(* Logix 5000 project; controller CLASE_1 Emulate 5570 rev 28.11; software revision 28.02; part 7 of 15 *)
(* tags used below, declared in another part *)
   Inp_OvrdCmd : DINT;   // Override Mode Command: 0=None, 1=Stop, 2=Start
   PCmd_Start : BOOL;   // Program Command to Start Motor
   PCmd_Stop : BOOL;   // Program Command to Stop Motor
   OCmd_Start : BOOL;   // Operator Command to Start Motor
   OCmd_Stop : BOOL;   // Operator Command to Stop Motor
   Out_Run : BOOL;   // 1=Run Motor, 0=Stop Motor
   Out_Start : BOOL;   // 1=Start Motor, 0=Motor left in current state
   Out_Stop : BOOL;   // 1=Stop Motor, 0=Motor left in current state
   Val_Cmd : SINT;   // Device Command 0=None, 1=Stop, 2=Start
   Nrdy_OperPrio : BOOL;   // 1=Device Not Ready: Operator State 0 Priority Command Requires Reset
   Nrdy_Fail : BOOL;   // 1=Device Not Ready: Device Failure (Shed Requires Reset)
   P_Motor : BOOL;   // Unique Parameter Name for auto - discovery
   Wrk_Run : BOOL;   // 1=Motor should be "running", 0=should be "stopped"
   Wrk_RunFdbk : BOOL;   // Run Feedback based on mode, simulation, etc. 1=running
(* P_Motor, continued *)

ROUTINE Prescan   (* ladder *)
// Clear Ownership, clear "lurking" Commands
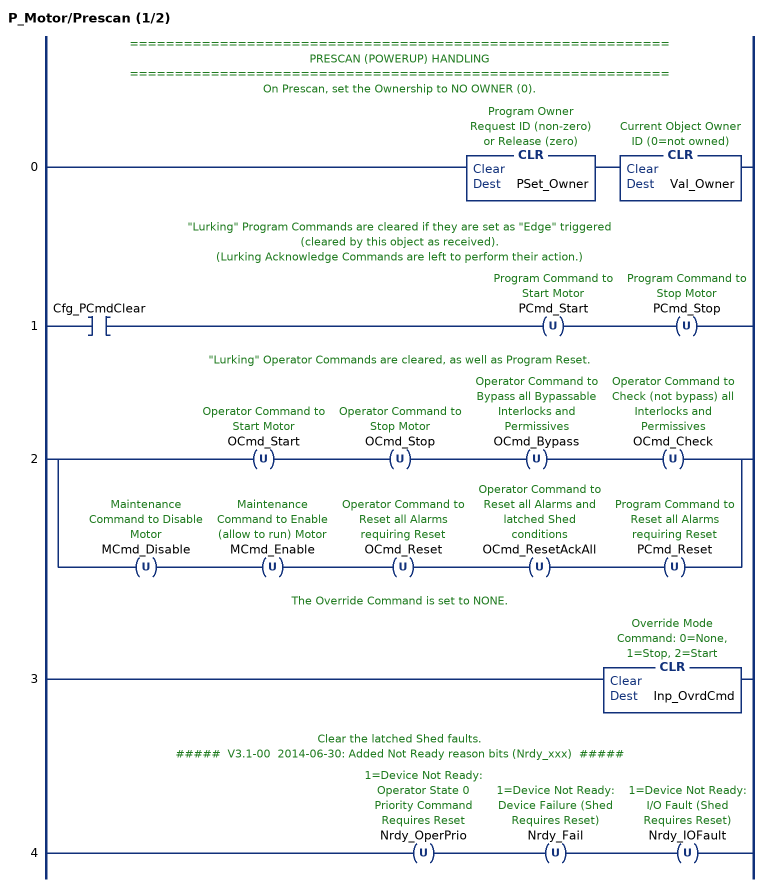
   // ============================================================
   // PRESCAN (POWERUP) HANDLING
   // ============================================================
   // On Prescan, set the Ownership to NO OWNER (0).
   0: CLR(PSet_Owner)CLR(Val_Owner);
   // "Lurking" Program Commands are cleared if they are set as "Edge" triggered
   // (cleared by this object as received).
   // (Lurking Acknowledge Commands are left to perform their action.)
   1: XIC(Cfg_PCmdClear)OTU(PCmd_Start)OTU(PCmd_Stop);
   // "Lurking" Operator Commands are cleared, as well as Program Reset.
   2: [OTU(OCmd_Start) OTU(OCmd_Stop) OTU(OCmd_Bypass) OTU(OCmd_Check) ,OTU(MCmd_Disable) OTU(MCmd_Enable) OTU(OCmd_Reset) OTU(OCmd_ResetAckAll) OTU(PCmd_Reset) ];
   // The Override Command is set to NONE.
   3: CLR(Inp_OvrdCmd);
   // Clear the latched Shed faults.
   // #####  V3.1-00  2014-06-30: Added Not Ready reason bits (Nrdy_xxx)  #####
   4: OTU(Nrdy_OperPrio)OTU(Nrdy_Fail)OTU(Nrdy_IOFault);
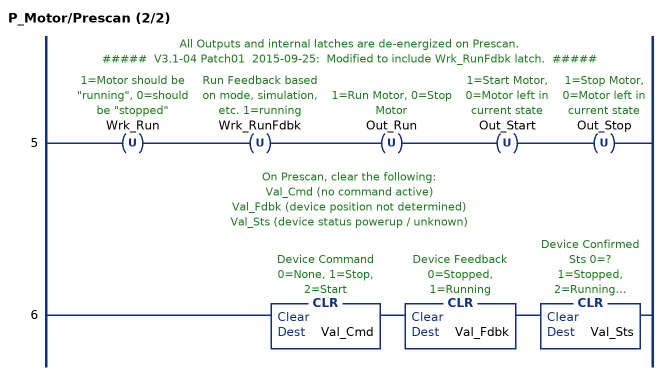
   // All Outputs and internal latches are de-energized on Prescan.
   // #####  V3.1-04 Patch01  2015-09-25:  Modified to include Wrk_RunFdbk latch.  #####
   5: OTU(Wrk_Run)OTU(Wrk_RunFdbk)OTU(Out_Run)OTU(Out_Start)OTU(Out_Stop);
   // On Prescan, clear the following:
   // Val_Cmd (no command active)
   // Val_Fdbk (device position not determined)
   // Val_Sts (device status powerup / unknown)
   6: CLR(Val_Cmd)CLR(Val_Fdbk)CLR(Val_Sts);
END_ROUTINE
END_ADD_ON_INSTRUCTION

ADD_ON_INSTRUCTION P_Perm   (* revision 3.5 05 Release, vendor Rockwell Automation, ExecutePrescan, ExecuteEnableInFalse *)
// Permissives
// Revision note:
// See V3.5-xx Release Notes for details. Changed Nav Tags to user-defined STRING_NavTag type.
// Help:
// Copyright © Rockwell Automation, Inc.  All Rights Reserved.
// This Instruction monitors up to 16 Permissive conditions.  It provides these features:
// *  The "OK" state of each Permissive Input is configurable.  By default,
//     each Input is 1 when OK to start, 0 when not OK to start.
// *  Permissives may be configured as Bypassable.  A separate Sts_NBPermOK
//     (Non-Bypassable Permissives OK) status is provided, which the destination
//     object can use for Bypass, Maintenance and other functions,
//     where Bypassable Permissives can be ignored.
// All Permissive Inputs must be in their configured "OK" states
// for the P_Perm instruction to provide a "PermOK" status.
// All non-bypassable Permissive inputs must be in their configured "OK" states
// for the P_Perm instruction to provide a "NBPermOK" status.
// For each Permissive condition, a Tag may be defined for navigation. Clicking
// the Permissive description will call up the associated Tag's Faceplate.
VAR_INPUT
   Inp_Perm00 : ALIAS FOR Wrk_Inp.0; {visible}   // Permissive Cond 00, OK to start if in configured OK state
   Inp_Perm01 : ALIAS FOR Wrk_Inp.1; {visible}   // Permissive Cond 01, OK to start if in configured OK state
   Inp_Perm02 : ALIAS FOR Wrk_Inp.2; {visible}   // Permissive Cond 02, OK to start if in configured OK state
   Inp_Perm03 : ALIAS FOR Wrk_Inp.3; {visible}   // Permissive Cond 03, OK to start if in configured OK state
   Inp_Perm04 : ALIAS FOR Wrk_Inp.4; {visible}   // Permissive Cond 04, OK to start if in configured OK state
   Inp_Perm05 : ALIAS FOR Wrk_Inp.5; {visible}   // Permissive Cond 05, OK to start if in configured OK state
   Inp_Perm06 : ALIAS FOR Wrk_Inp.6; {visible}   // Permissive Cond 06, OK to start if in configured OK state
   Inp_Perm07 : ALIAS FOR Wrk_Inp.7; {visible}   // Permissive Cond 07, OK to start if in configured OK state
   Inp_Perm08 : ALIAS FOR Wrk_Inp.8;   // Permissive Cond 08, OK to start if in configured OK state
   Inp_Perm09 : ALIAS FOR Wrk_Inp.9;   // Permissive Cond 09, OK to start if in configured OK state
   Inp_Perm10 : ALIAS FOR Wrk_Inp.10;   // Permissive Cond 10, OK to start if in configured OK state
   Inp_Perm11 : ALIAS FOR Wrk_Inp.11;   // Permissive Cond 11, OK to start if in configured OK state
   Inp_Perm12 : ALIAS FOR Wrk_Inp.12;   // Permissive Cond 12, OK to start if in configured OK state
   Inp_Perm13 : ALIAS FOR Wrk_Inp.13;   // Permissive Cond 13, OK to start if in configured OK state
   Inp_Perm14 : ALIAS FOR Wrk_Inp.14;   // Permissive Cond 14, OK to start if in configured OK state
   Inp_Perm15 : ALIAS FOR Wrk_Inp.15;   // Permissive Cond 15, OK to start if in configured OK state
   Inp_BypActive : BOOL; {visible}   // 1=Permissive Bypassing is currently active
   Cfg_OKState : INT := 2#1111_1111_1111_1111;   // Bits indicate which state (0 or 1) of each input is OK to start
   Cfg_Bypassable : INT;   // Set bits indicate which conditions can be bypassed
   Cfg_HasNav : INT;   // Set bits indicate which Navigation buttons are enabled
   MSet_Bypass00 : ALIAS FOR Wrk_MSet.0;   // Maint. Bypass Toggle for Interlock Cond. 00: 1=Bypass
   MSet_Bypass01 : ALIAS FOR Wrk_MSet.1;   // Maint. Bypass Toggle for Interlock Cond. 0`: 1=Bypass
   MSet_Bypass02 : ALIAS FOR Wrk_MSet.2;   // Maint. Bypass Toggle for Interlock Cond. 02: 1=Bypass
   MSet_Bypass03 : ALIAS FOR Wrk_MSet.3;   // Maint. Bypass Toggle for Interlock Cond. 03: 1=Bypass
   MSet_Bypass04 : ALIAS FOR Wrk_MSet.4;   // Maint. Bypass Toggle for Interlock Cond. 04: 1=Bypass
   MSet_Bypass05 : ALIAS FOR Wrk_MSet.5;   // Maint. Bypass Toggle for Interlock Cond. 05: 1=Bypass
   MSet_Bypass06 : ALIAS FOR Wrk_MSet.6;   // Maint. Bypass Toggle for Interlock Cond. 06: 1=Bypass
   MSet_Bypass07 : ALIAS FOR Wrk_MSet.7;   // Maint. Bypass Toggle for Interlock Cond. 07: 1=Bypass
   MSet_Bypass08 : ALIAS FOR Wrk_MSet.8;   // Maint. Bypass Toggle for Interlock Cond. 08: 1=Bypass
   MSet_Bypass09 : ALIAS FOR Wrk_MSet.9;   // Maint. Bypass Toggle for Interlock Cond. 09: 1=Bypass
   MSet_Bypass10 : ALIAS FOR Wrk_MSet.10;   // Maint. Bypass Toggle for Interlock Cond. 10: 1=Bypass
   MSet_Bypass11 : ALIAS FOR Wrk_MSet.11;   // Maint. Bypass Toggle for Interlock Cond. 11: 1=Bypass
   MSet_Bypass12 : ALIAS FOR Wrk_MSet.12;   // Maint. Bypass Toggle for Interlock Cond. 12: 1=Bypass
   MSet_Bypass13 : ALIAS FOR Wrk_MSet.13;   // Maint. Bypass Toggle for Interlock Cond. 13: 1=Bypass
   MSet_Bypass14 : ALIAS FOR Wrk_MSet.14;   // Maint. Bypass Toggle for Interlock Cond. 14: 1=Bypass
   MSet_Bypass15 : ALIAS FOR Wrk_MSet.15;   // Maint. Bypass Toggle for Interlock Cond. 15: 1=Bypass
END_VAR
VAR_OUTPUT
   Sts_PermOK : BOOL := 1; {access Read Only, visible}   // Overall Permissive Status (1=OK to start)
   Sts_NBPermOK : BOOL := 1; {access Read Only, visible}   // Non-Bypassable Permissive Status (1 =all non- bypassable Permissives OK to start)
   Sts_BypActive : BOOL; {access Read Only}   // 1=Permissive Bypassing is Active (ignore bypassable permissives)
   Sts_Perm : INT := 2#1111_1111_1111_1111; {access Read Only, visible}   // Individual Permissive Status (1=OK, 0=don't start)
   P_Perm : BOOL;   // Unique Parameter Name for auto - discovery
END_VAR
VAR
   Cfg_CondTxt : STRING_20[16] := ([0] := 'Enter Description #0');   // Short HMI description of Permissive Conditions
   Wrk_Inp : INT := 2#1111_1111_1111_1111;   // Collection copy of Inp_PermXXs
   Wrk_Bypass : INT; {access None}   // Working Register for Bypassable Permissives
   Inf_Tab : SINT;   // Tab to display (FTView ME)
   Wrk_InpInv : INT; {access None}   // Input states after inverting based on Cfg_OKState
   Inf_Type : STRING_16 := 'P_Perm'; {access Read Only}   // Type identifier for HMI navigation
   Cfg_Label : STRING_20 := 'Permissives';   // Label for graphic symbol displayed on HMI
   Cfg_Tag : STRING_20 := 'P_Perm';   // Tagname for display on HMI
   Cfg_Desc : STRING_40 := 'Permissives';   // Description for display on HMI
   Cfg_NavTag : STRING_NavTag[16];   // Tagnames for destinations of Navigation buttons
   Inf_Lib : STRING_12 := 'RA-BAS'; {access Read Only}   // Display Library for Faceplate call-up
   Wrk_MSet : INT;   // Internal copy of individual condition Maint. Bypass toggles
END_VAR

ROUTINE EnableInFalse   (* ladder *)
// Set summary "OK" Status bits to FALSE (0)
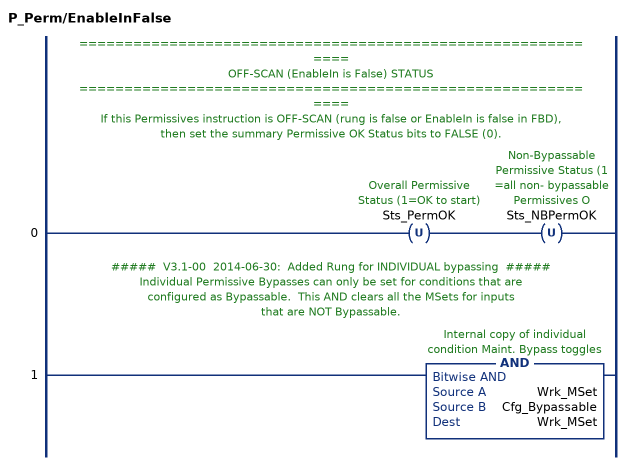
   // ============================================================
   // OFF-SCAN (EnableIn is False) STATUS
   // ============================================================
   // If this Permissives instruction is OFF-SCAN (rung is false or EnableIn is false in FBD),
   // then set the summary Permissive OK Status bits to FALSE (0).
   0: OTU(Sts_PermOK)OTU(Sts_NBPermOK);
   // #####  V3.1-00  2014-06-30:  Added Rung for INDIVIDUAL bypassing  #####
   // Individual Permissive Bypasses can only be set for conditions that are
   // configured as Bypassable.  This AND clears all the MSets for inputs
   // that are NOT Bypassable.
   1: AND(Wrk_MSet,Cfg_Bypassable,Wrk_MSet);
END_ROUTINE

ROUTINE Logic   (* ladder *)
// Check Permissive Conditions
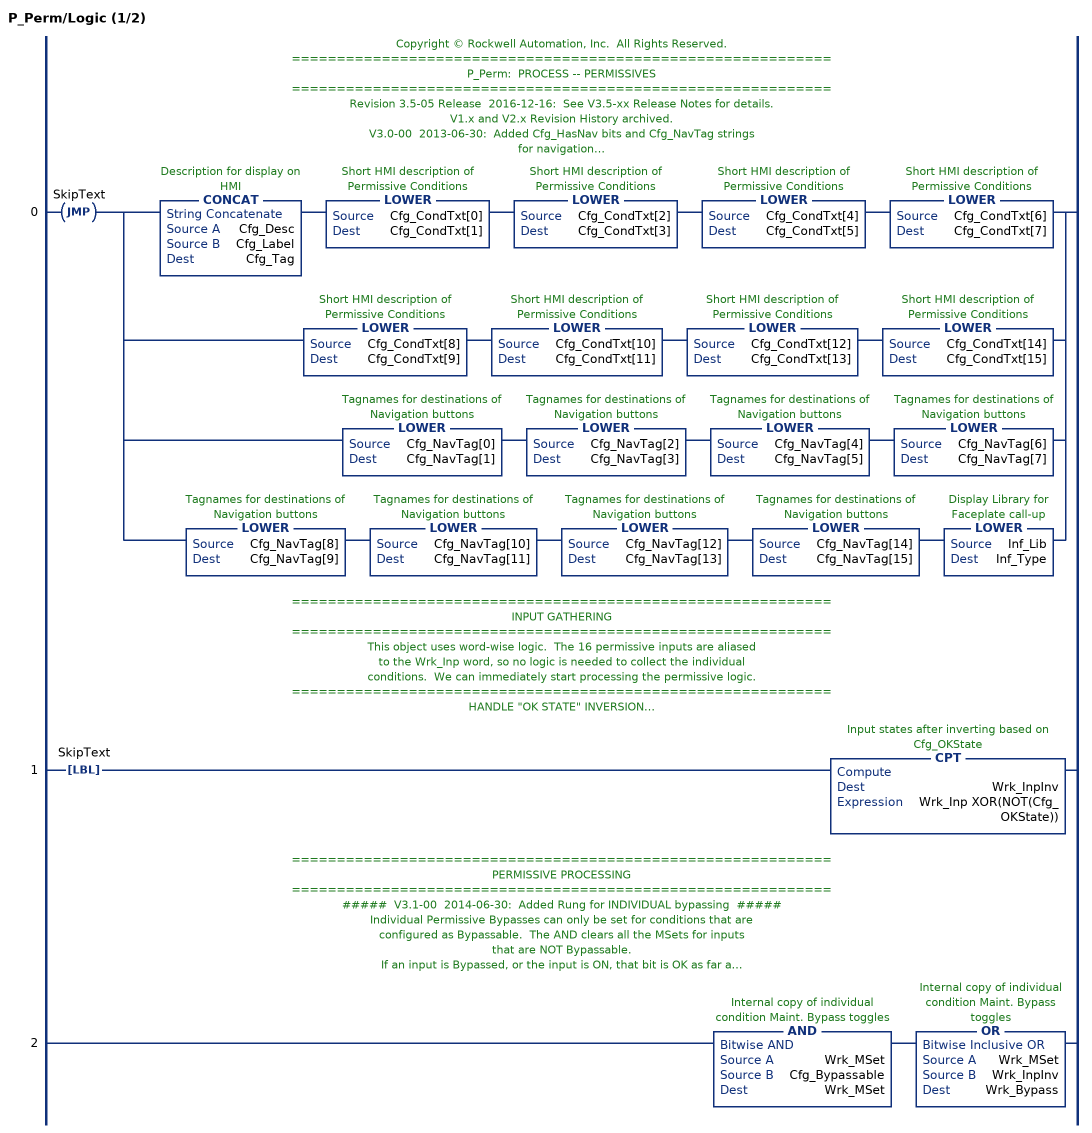
   // Copyright © Rockwell Automation, Inc.  All Rights Reserved.
   // ============================================================
   // P_Perm:  PROCESS -- PERMISSIVES
   // ============================================================
   // Revision 3.5-05 Release  2016-12-16:  See V3.5-xx Release Notes for details.
   // V1.x and V2.x Revision History archived.
   // V3.0-00  2013-06-30:  Added Cfg_HasNav bits and Cfg_NavTag strings
   // for navigation.
   // V3.1-00  2014-06-30:  Modified to allow Maintenance to set up bypassing
   // of individual permissive conditions.
   // V3.1-01  2014-09-03:  Unmodified, up-rev only for V3.1-01 public release.
   // V3.5-01  2016-01-29:  Unmodified, up-rev only for V3.5-01 Release.
   // V3.5-05  2016-12-16:  Changed Nav Tags to user-defined STRING_NavTag type.
   // ============================================================
   // This Instruction monitors up to 16 Permissive conditions.  It provides these features:
   // *  The "OK" state of each Permissive Input is configurable.  By default,
   // each Input is 1 when OK to start, 0 when not OK to start.
   // *  Permissives may be configured as Bypassable.  A separate Sts_NBPermOK
   // (Non-Bypassable Permissives OK) status is provided, which the destination
   // object can use forBypass, Maintenance and other functions,
   // where Bypassable Permissives can be ignored.
   // All Permissive Inputs must be in their configured "OK" states
   // for the P_Perm instruction to provide a "PermOK" status.
   // All non-bypassable Permissive inputs must be in their configured "OK" states
   // for the P_Perm instruction to provide a "NBPermOK" status.
   // For each Permissive condition, a Tag may be defined for navigation. Clicking
   // the Permissive description will call up the associated Tag's Faceplate.
   // ============================================================
   // SHOW LOCAL STRINGS
   // ============================================================
   // The STRINGs containing the text associated with each instance of this
   // instruction cannot be Input or Output Parameters, because STRINGs are not
   //  'atomic' types. (Inputs and Outputs must be SINT, INT, DINT, REAL, or BOOL.)
   // In order to make it easier to find and configure these STRINGs, this rung
   // was added.  THE JMP (and the LBL on the following rung)
   // MUST NOT BE REMOVED!!!
   // To view the STRINGs, go to the instruction instance (in LD or FBD), RIGHT-click
   // to bring up the context menu and select "Open Instruction Logic".
   // This rung will appear with the STRING values for the selected instance.
   // You may double-click the STRING values here to modify them as well.
   // #####  V3.0-00  2013-06-30:  Added Cfg_NavTag strings on this rung  #####
   0: JMP(SkipText)[CONCAT(Cfg_Desc,Cfg_Label,Cfg_Tag) LOWER(Cfg_CondTxt[0],Cfg_CondTxt[1]) LOWER(Cfg_CondTxt[2],Cfg_CondTxt[3]) LOWER(Cfg_CondTxt[4],Cfg_CondTxt[5]) LOWER(Cfg_CondTxt[6],Cfg_CondTxt[7]) ,LOWER(Cfg_CondTxt[8],Cfg_CondTxt[9]) LOWER(Cfg_CondTxt[10],Cfg_CondTxt[11]) LOWER(Cfg_CondTxt[12],Cfg_CondTxt[13]) LOWER(Cfg_CondTxt[14],Cfg_CondTxt[15]) ,LOWER(Cfg_NavTag[0],Cfg_NavTag[1]) LOWER(Cfg_NavTag[2],Cfg_NavTag[3]) LOWER(Cfg_NavTag[4],Cfg_NavTag[5]) LOWER(Cfg_NavTag[6],Cfg_NavTag[7]) ,LOWER(Cfg_NavTag[8],Cfg_NavTag[9]) LOWER(Cfg_NavTag[10],Cfg_NavTag[11]) LOWER(Cfg_NavTag[12],Cfg_NavTag[13]) LOWER(Cfg_NavTag[14],Cfg_NavTag[15]) LOWER(Inf_Lib,Inf_Type) ];
   // ============================================================
   // INPUT GATHERING
   // ============================================================
   // This object uses word-wise logic.  The 16 permissive inputs are aliased
   // to the Wrk_Inp word, so no logic is needed to collect the individual
   // conditions.  We can immediately start processing the permissive logic.
   // ============================================================
   // HANDLE "OK STATE" INVERSIONS
   // ============================================================
   // This rung inverts the Input bits whose "OK State" is 1 (0 to Run).
   // The resulting Wrk_Inp word is ALL ONES if all permissive inputs are "OK".
   1: LBL(SkipText)CPT(Wrk_InpInv,Wrk_Inp XOR(NOT(Cfg_OKState)));
   // ============================================================
   // PERMISSIVE PROCESSING
   // ============================================================
   // #####  V3.1-00  2014-06-30:  Added Rung for INDIVIDUAL bypassing  #####
   // Individual Permissive Bypasses can only be set for conditions that are
   // configured as Bypassable.  The AND clears all the MSets for inputs
   // that are NOT Bypassable.
   // If an input is Bypassed, or the input is ON, that bit is OK as far as
   // Bypassable Permissives are concerned.
   2: AND(Wrk_MSet,Cfg_Bypassable,Wrk_MSet)OR(Wrk_MSet,Wrk_InpInv,Wrk_Bypass);
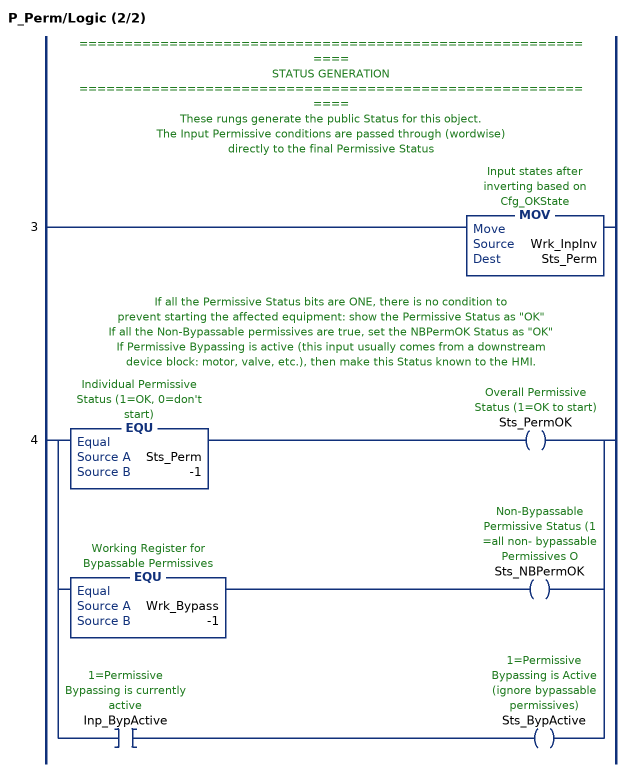
   // ============================================================
   // STATUS GENERATION
   // ============================================================
   // These rungs generate the public Status for this object.
   // The Input Permissive conditions are passed through (wordwise)
   // directly to the final Permissive Status
   3: MOV(Wrk_InpInv,Sts_Perm);
   // If all the Permissive Status bits are ONE, there is no condition to
   // prevent starting the affected equipment: show the Permissive Status as "OK"
   // If all the Non-Bypassable permissives are true, set the NBPermOK Status as "OK"
   // If Permissive Bypassing is active (this input usually comes from a downstream
   // device block: motor, valve, etc.), then make this Status known to the HMI.
   4: [EQU(Sts_Perm,-1) OTE(Sts_PermOK) ,EQU(Wrk_Bypass,-1) OTE(Sts_NBPermOK) ,XIC(Inp_BypActive) OTE(Sts_BypActive) ];
END_ROUTINE

ROUTINE Prescan   (* ladder *)
// On powerup, clear individual bypass enables for non-bypassable permissives.
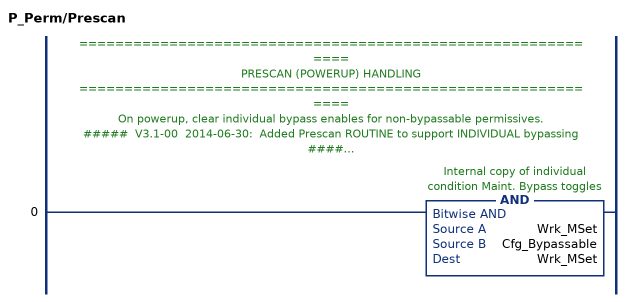
   // ============================================================
   // PRESCAN (POWERUP) HANDLING
   // ============================================================
   // On powerup, clear individual bypass enables for non-bypassable permissives.
   // #####  V3.1-00  2014-06-30:  Added Prescan ROUTINE to support INDIVIDUAL bypassing  #####
   // Individual Permissive Bypasses can only be set for conditions that are
   // configured as Bypassable.  This AND clears all the MSets for inputs
   // that are NOT Bypassable.
   0: AND(Wrk_MSet,Cfg_Bypassable,Wrk_MSet);
END_ROUTINE
END_ADD_ON_INSTRUCTION

ADD_ON_INSTRUCTION P_ValveC   (* revision 3.5 08 Release, vendor Rockwell Automation, ExecutePrescan, ExecuteEnableInFalse *)
// Control Valve
// Revision note:
// See V3.5-xx Release Notes for details. Modified CV Rate of Change handling for limits = 0.0 (unlimited).
// Help:
// Copyright © Rockwell Automation, Inc.  All Rights Reserved.
// This Instruction controls a Pulse Output Valve with analog position feedback and provides:
// *  Program and Operator entry of target position in Percent Open
// *  Ramping of position to target at specified Rate of Change (%/sec)
// *  Scaling of Position Feedback input from Raw (I/O card) Units to percent
// *  Monitoring of Interlock conditions which cause output to shed
// *  Configurable shed to HOLD or to configured position
// *  Monitoring of I/O communication faults
// *  Alarms for Interlock Trip, Actuator Fault, I/O Fault
// *  Operation in Hand, Maintenance, Override, Program and Operator Modes
// *  "Available" status for use by automation logic to know whether valve
//       can be controlled by other objects.
// Modes are provided by a P_Mode AOI instance.
// Alarms are provided by P_Alarm AOI instances.
// Modes of operation: Operator, Program, Override, Maintenance, Hand
// Configuration notes:
//    If Max ON Time is less than 0 or greater than the Cycle Time
//         it is set to the Cycle Time.
//    If Min ON Time is less than 0 or greater than the Max ON Time
//         it is set to zero.
//    If Deadtime is less than 0 or greater than the Cycle Time,
//         it is set to zero.
//    Bump Time must be within the Min ON Time and Max ON Time.
VAR_INPUT
   Inp_PosFdbk : REAL; {visible}   // Position Feedback from Valve (in Raw Input units)
   Inp_OpenLS : BOOL; {visible}   // Valve Open Limit Switch 1=confirmed fully open
   Inp_ClosedLS : BOOL; {visible}   // Valve Closed Limit Switch 1=confirmed fully closed
   Inp_ActuatorFault : BOOL; {visible}   // Valve Actuator Fault (overload, etc.), 0=OK, 1=Fault)
   Inp_IntlkOK : BOOL := 1; {visible}   // 1=Interlocks OK, Pulse Output Valve can be moved
   Inp_NBIntlkOK : BOOL := 1; {visible}   // 1=Non-Bypassable Interlocks OK, Pulse Output Valve can be moved
   Inp_IOFault : BOOL;   // Input / Output Communication Status 0=OK, 1=fail
   Inp_Sim : BOOL;   // 1=I/O are being simulated, set output CV to 0.0, ignore I/O Fault
   Inp_Hand : ALIAS FOR Mode.Inp_Hand;
   Inp_Ovrd : ALIAS FOR Mode.Inp_Ovrd;
   Inp_OvrdCV : REAL;   // CV target in Override Mode (CV EU)
   Inp_Reset : BOOL;   // 1=Reset latched Alarms
   Cfg_ShedHold : BOOL;   // 1=Hold Output on Interlock or bad PV, 0=Go to Cfg_IntlkCV
   Cfg_ShedOnIOFault : BOOL := 1;   // 1=Take shed action (hold or interlock CV) on I/O Fault
   Cfg_SkipRoCLim : BOOL;   // 1=Skip RoC Limiting in Intlk, Maint, Ovrd modes
   Cfg_SetTrack : BOOL := 1;   // 1=PSets track OSets in Oper, OSets track PSets in Prog, 0=no tracking
   Cfg_SetTrackOvrdHand : BOOL;   // 1=Prog/Oper Settings track Override/Hand CV
   Cfg_HasOpenLS : BOOL;   // 1=Valve provides an Open Limit Switch signal
   Cfg_HasClosedLS : BOOL;   // 1=Valve provides a Closed Limit Switch signal
   Cfg_UseOpenLS : BOOL;   // 1=Valve Open LS should be used for open/closed status
   Cfg_UseClosedLS : BOOL;   // 1=Valve Closed LS should be used for open/closed status
   Cfg_LSFail : BOOL := 1;   // 1=both switches ON=fail, 0=both switches OFF=fail
   Cfg_HasIntlkObj : BOOL;   // 1=Tells HMI a P_Intlk is connected to Inp_Intlk
   Cfg_HasCVNav : BOOL;   // 1=Tells HMI to enable navigation to a connected CV object
   Cfg_PCmdClear : ALIAS FOR Mode.Cfg_PCmdClear;
   Cfg_ProgDefault : ALIAS FOR Mode.Cfg_ProgDefault;
   Cfg_OvrdIntlk : BOOL;   // 1=Override ignores Bypassable Intlk; 0=always use Intlk
   Cfg_HasIntlkTripAlm : ALIAS FOR IntlkTrip.Cfg_Exists;   // 1=Interlock Trip Alarm exists and will be checked
   Cfg_HasActuatorFaultAlm : ALIAS FOR ActuatorFault.Cfg_Exists;   // 1=Actuator Fault Alarm exists and will be checked
   Cfg_HasIOFaultAlm : ALIAS FOR IOFault.Cfg_Exists;   // 1=I/O Fault Alarm exists and will be checked
   Cfg_IntlkTripResetReqd : ALIAS FOR IntlkTrip.Cfg_ResetReqd;   // 1=Reset required to clear Interlock Trip Alarm
   Cfg_ActuatorFaultResetReqd : ALIAS FOR ActuatorFault.Cfg_ResetReqd;   // 1=Reset required to clear Actuator Fault Alarm
   Cfg_IOFaultResetReqd : ALIAS FOR IOFault.Cfg_ResetReqd;   // 1=Reset required to clear I/O Fault Alarm
   Cfg_IntlkTripAckReqd : ALIAS FOR IntlkTrip.Cfg_AckReqd;   // 1=Acknowledge required for Interlock Trip Alarm
   Cfg_ActuatorFaultAckReqd : ALIAS FOR ActuatorFault.Cfg_AckReqd;   // 1=Acknowledge required for Actuator Fault Alarm
   Cfg_IOFaultAckReqd : ALIAS FOR IOFault.Cfg_AckReqd;   // 1=Acknowledge required for I/O Fault Alarm
   Cfg_IntlkTripSeverity : ALIAS FOR IntlkTrip.Cfg_Severity;   // Interlock Trip Alarm Severity: 1..250=Low, 251..500=Medium, 501..750=High, 751..1000=Urgent
   Cfg_ActuatorFaultSeverity : ALIAS FOR ActuatorFault.Cfg_Severity;   // Actuator Fault Alarm Severity: 1..250=Low, 251..500=Medium, 501..750=High, 751..1000=Urgent
   Cfg_IOFaultSeverity : ALIAS FOR IOFault.Cfg_Severity;   // I/O Fault Alarm Severity: 1..250=Low, 251..500=Medium, 501..750=High, 751..1000=Urgent
   Cfg_MinCV : REAL;   // Minimum CV (in CV EU, for limiting)
   Cfg_MaxCV : REAL := 100.0;   // Maximum CV (in CV EU, for limiting)
   Cfg_MaxCVRoCInc : REAL := 10.0;   // Maximum allowed CV Rate of Change (Increasing) Setting (EU/sec)
   Cfg_MaxCVRoCDec : REAL := 10.0;   // Maximum allowed CV Rate of Change (Decreasing) Setting (EU/sec)
   Cfg_IntlkCV : REAL;   // CV (target in EU) when interlocked (if not Cfg_ShedHold)
   Cfg_CVEUMin : REAL;   // CV Minimum in Engineering Units (for scaling)
   Cfg_CVEUMax : REAL := 100.0;   // CV Maximum in Engineering Units (for scaling)
   Cfg_CVRawMin : REAL;   // CV Minimum in I/O (raw) Units (for scaling)
   Cfg_CVRawMax : REAL := 100.0;   // CV Maximum in I/O (raw) Units (for scaling)
   Cfg_FdbkRawMin : REAL;   // Position Feedback Minimum in raw input units (for scaling)
   Cfg_FdbkRawMax : REAL := 100.0;   // Position Feedback Maximum in raw input units (for scaling)
   Cfg_CycleT : REAL := 10.0;   // Open and Close Pulse Output overall period (s)
   Cfg_OpenRate : REAL := 1.0;   // Rate at which valve moves when opening (CV EU/sec)
   Cfg_CloseRate : REAL := 1.0;   // Rate at which valve moves when closing (CV EU/sec)
   Cfg_MaxOnT : REAL := 5.0;   // Open and Close Pulse Output maximum ON time (s)
   Cfg_MinOnT : REAL := 1.0;   // Open and Close Pulse Output minimum ON time (s)
   Cfg_BumpT : REAL;   // Time to bump valve open or closed (by Oper) when Fdbk Bad (sec)
   Cfg_Deadtime : REAL;   // Additional time on first pulse after stop or direction change
   Cfg_MaxClosedPos : REAL;   // Position above which valve is assumed open if limit switches not used
   PSet_CV : REAL;   // Program Setting of Controlled Variable (output) (CV EU)
   PSet_CVRoCLimInc : REAL;   // Program Setting of CV Rate of Change Limit, Increasing, (in EU/sec)
   PSet_CVRoCLimDec : REAL;   // Program Setting of CV Rate of Change Limit, Decreasing, (in EU/sec)
   PSet_Owner : DINT;   // Program Owner Request ID (non-zero) or Release (zero)
   OSet_CV : REAL;   // Operator Setting of Controlled Variable (output) (CV EU)
   OSet_CVRoCLimInc : REAL;   // Operator Setting of CV Rate of Change Limit, Increasing, (in EU/sec)
   OSet_CVRoCLimDec : REAL;   // Operator Setting of CV Rate of Change Limit, Decreasing, (in EU/sec)
   PCmd_Acq : ALIAS FOR Mode.PCmd_Acq;
   PCmd_Rel : ALIAS FOR Mode.PCmd_Rel;
   PCmd_Lock : ALIAS FOR Mode.PCmd_Lock;
   PCmd_Unlock : ALIAS FOR Mode.PCmd_Unlock;
   PCmd_Reset : BOOL;   // Program Command to Reset Alarms requiring Reset
   PCmd_IntlkTripAck : ALIAS FOR IntlkTrip.PCmd_Ack;   // Program Command to Acknowledge Interlock Trip Alarm
   PCmd_IntlkTripSuppress : ALIAS FOR IntlkTrip.PCmd_Suppress;   // Program Command to Suppress Interlock Trip Alarm
   PCmd_IntlkTripUnsuppress : ALIAS FOR IntlkTrip.PCmd_Unsuppress;   // Program Command to Unsuppress Interlock Trip Alarm
   PCmd_IntlkTripUnshelve : ALIAS FOR IntlkTrip.PCmd_Unshelve;   // Program Command to Unshelve Interlock Trip Alarm
   PCmd_ActuatorFaultAck : ALIAS FOR ActuatorFault.PCmd_Ack;   // Program Command to Acknowledge Actuator Fault Alarm
   PCmd_ActuatorFaultSuppress : ALIAS FOR ActuatorFault.PCmd_Suppress;   // Program Command to Suppress Actuator Fault Alarm
   PCmd_ActuatorFaultUnsuppress : ALIAS FOR ActuatorFault.PCmd_Unsuppress;   // Program Command to Unsuppress Actuator Fault Alarm
   PCmd_ActuatorFaultUnshelve : ALIAS FOR ActuatorFault.PCmd_Unshelve;   // Program Command to Unshelve Actuator Fault Alarm
   PCmd_IOFaultAck : ALIAS FOR IOFault.PCmd_Ack;   // Program Command to Acknowledge I/O Fault Alarm
   PCmd_IOFaultSuppress : ALIAS FOR IOFault.PCmd_Suppress;   // Program Command to Suppress I/O Fault Alarm
   PCmd_IOFaultUnsuppress : ALIAS FOR IOFault.PCmd_Unsuppress;   // Program Command to Unsuppress I/O Fault Alarm
   PCmd_IOFaultUnshelve : ALIAS FOR IOFault.PCmd_Unshelve;   // Program Command to Unshelve I/O Fault Alarm
   OCmd_BumpOpen : BOOL;   // Operator Command to bump valve open (avail. if Fdbk Bad)
   OCmd_BumpClose : BOOL;   // Operator Command to bump valve closed (avail. if Fdbk Bad)
   OCmd_Bypass : BOOL;   // Operator Command to Bypass all Bypassable Interlocks
   OCmd_Check : BOOL;   // Operator Command to Check (not bypass) all Interlocks
   MCmd_Disable : BOOL;   // Maintenance Command to Pulse Output Valve
   MCmd_Enable : BOOL;   // Maintenance Command to Enable Pulse Output Valve
   MCmd_Acq : ALIAS FOR Mode.MCmd_Acq;
   MCmd_Rel : ALIAS FOR Mode.MCmd_Rel;
   OCmd_AcqLock : ALIAS FOR Mode.OCmd_AcqLock;
   OCmd_Unlock : ALIAS FOR Mode.OCmd_UnlockRel;
   OCmd_Reset : BOOL;   // Operator Command to Reset all Alarms requiring Reset
   OCmd_ResetAckAll : BOOL;   // Operator Command to Reset all Alarms and latched Shed conditions
END_VAR
VAR_OUTPUT
   Out_CV : REAL; {access Read Only, visible}   // CV Output in Raw (I/O Card) Units
   Out_Open : BOOL; {access Read Only, visible}   // Pulse Output to drive valve Open
   Out_Close : BOOL; {access Read Only, visible}   // Pulse Output to drive valve closed
   Val_Pos : REAL; {access Read Only, visible}   // Valve actual position from feedback (CV EU)
   Val_CVSet : REAL; {access Read Only, visible}   // Value of selected CV Setting (before rate limiting, CV EU)
   Val_CVOut : REAL; {access Read Only, visible}   // Value of CV output (after clamping and ramping) (CV EU)
   Val_CVRoCLimInc : REAL; {access Read Only, visible}   // Value of CV Rate of Change Limit, Increasing, (in EU/sec)
   Val_CVRoCLimDec : REAL; {access Read Only, visible}   // Value of CV Rate of Change Limit, Decreasing, (in EU/sec)
   Val_CVEUMin : REAL; {access Read Only, visible}   // Minimum of scaled range = MIN (Cfg_CVEUMin, Cfg_CVEUMax)
   Val_CVEUMax : REAL := 100.0; {access Read Only, visible}   // Maximum of scaled range = MAX (Cfg_CVEUMin, Cfg_CVEUMax)
   SrcQ_IO : SINT; {access Read Only}   // Source and Quality of primary I/O (enumeration)
   SrcQ : SINT; {access Read Only}   // Source and Quality of primary Val/Sts (enumeration)
   Val_Fdbk : SINT; {access Read Only}   // Device Feedback 0=Moving, 1=Closed, 2=Opened, 3=Limit Switch Failure
   Val_Sts : SINT; {access Read Only}   // 0=AtTarget, 1=RampClose, 2=RampOpen, 3=Clamp@Min, 4=Clamp@Max, 5=BumpClose, 6=BumpOpen, 33=Disabled
   Val_Fault : SINT; {access Read Only}   // Device Fault Status 0=none, 32=I/OFault, 34=CfgErr
   Val_Mode : ALIAS FOR Mode.Val; {access Read Only}
   Val_Owner : DINT; {access Read Only}   // Current Object Owner ID (0=not owned)
   Val_Notify : SINT; {access Read Only}   // Current Alarm Level and Acknowledgement (enumeration)
   Sts_CVInfNaN : BOOL; {access Read Only}   // 1=Selected CV is Infinite or Not A Number (1.$, 1.#NaN)
   Sts_PosInfNaN : BOOL; {access Read Only}   // 1=Inp_PosFdbk is Infinite or Not A Number (1.$, 1.#NaN)
   Sts_BumpOpen : BOOL; {access Read Only}   // 1=Bump Open Requested or Active
   Sts_BumpClose : BOOL; {access Read Only}   // 1=Bump Close Requested or Active
   Sts_Ramping : BOOL; {access Read Only}   // 1=CV is ramping to target
   Sts_Clamped : BOOL; {access Read Only}   // 1=CV Set is clamped at CVMin or CVMax
   Sts_SkipRoCLim : BOOL; {access Read Only}   // 1=Rate of Change Limiting was skipped this scan (Maint, Ovrd, Intlk, Hand)
   Sts_Active : BOOL; {access Read Only}   // 1=CV is greater than Cfg_MaxClosedPos, show valve symbol as "opened"
   Sts_Available : BOOL; {access Read Only}   // 1=Pulse Output Valve available for control by automation (Prog)
   Sts_Bypass : BOOL; {access Read Only}   // 1=Bypassable Interlocks are Bypassed
   Sts_BypActive : BOOL; {access Read Only}   // 1=Bypassing Active (Bypassed or Maintenance)
   Sts_Disabled : BOOL; {access Read Only}   // 1=Output is Disabled
   Sts_LSFail : BOOL; {access Read Only}   // 1=Limit Switch Overlap Failure
   Sts_NotRdy : BOOL; {access Read Only}   // 1=Device Not Ready, see detail bits for reason
   Nrdy_Disabled : BOOL; {access Read Only}   // 1=Device Not Ready: Device Disabled by Maintenance
   Nrdy_CfgErr : BOOL; {access Read Only}   // 1=Device Not Ready: Configuration Error
   Nrdy_Intlk : BOOL; {access Read Only}   // 1=Device Not Ready: Interlock Not OK
   Nrdy_IOFault : BOOL; {access Read Only}   // 1=Device Not Ready: I/O Fault (Shed Requires Reset)
   Nrdy_NoMode : BOOL; {access Read Only}   // 1=Device Not Ready: Device Logic Disabled / NO Mode
   Sts_MaintByp : BOOL; {access Read Only}   // 1=Device has a Maintenance Bypass function active
   Sts_AlmInh : BOOL; {access Read Only}   // 1=One or more Alarms Shelved, Disabled or Suppressed
   Sts_Err : BOOL; {access Read Only, visible}   // 1=Error in Config: see detail bits for reason
   Err_Limit : BOOL; {access Read Only}   // 1=Error in Config: CV Limits swapped
   Err_EU : BOOL; {access Read Only}   // 1=Error in Config: Scaled CV EU Min = Max
   Err_Raw : BOOL; {access Read Only}   // 1=Error in Config: Raw Output Scaling Min = Max
   Err_Fdbk : BOOL; {access Read Only}   // 1=Error in Config: Raw Feedback Scaling Min = Max
   Err_Timer : BOOL; {access Read Only}   // 1=Error in Config: Invalid Timer Preset (use 0 to 2147483)
   Err_Alarm : BOOL; {access Read Only}   // 1=Error in Config: Alarm Min On Time, Shelf Time, Severity
   Sts_Hand : ALIAS FOR Mode.Sts_Hand; {access Read Only, visible}
   Sts_Maint : ALIAS FOR Mode.Sts_Maint; {access Read Only, visible}
   Sts_Ovrd : ALIAS FOR Mode.Sts_Ovrd; {access Read Only, visible}
   Sts_Prog : ALIAS FOR Mode.Sts_Prog; {access Read Only, visible}
   Sts_Oper : ALIAS FOR Mode.Sts_Oper; {access Read Only, visible}
   Sts_ProgOperLock : ALIAS FOR Mode.Sts_ProgOperLock; {access Read Only}
   Sts_NoMode : ALIAS FOR Mode.Sts_NoMode; {access Read Only}
   Sts_MAcqRcvd : ALIAS FOR Mode.Sts_MAcqRcvd; {access Read Only}
   Sts_IntlkTrip : ALIAS FOR IntlkTrip.Inp;   // 1=Status: CV held or forced by interlock NOT OK (1-shot)
   Alm_IntlkTrip : ALIAS FOR IntlkTrip.Alm;   // 1=Alarm: CV held or forced by interlock NOT OK
   Ack_IntlkTrip : ALIAS FOR IntlkTrip.Ack;   // 1=Interlock Trip Alarm has been acknowledged
   Sts_IntlkTripDisabled : ALIAS FOR IntlkTrip.Disabled;   // 1=Interlock Trip Alarm has been Disabled by Maintenance
   Sts_IntlkTripShelved : ALIAS FOR IntlkTrip.Shelved;   // 1=Interlock Trip Alarm has been Shelved by Operator
   Sts_IntlkTripSuppressed : ALIAS FOR IntlkTrip.Suppressed;   // 1=Interlock Trip Alarm has been Suppressed by Program
   Sts_ActuatorFault : ALIAS FOR ActuatorFault.Inp;   // 1=Actuator Fault detected (input)
   Alm_ActuatorFault : ALIAS FOR ActuatorFault.Alm;   // 1=Alarm: Actuator Fault Detected
   Ack_ActuatorFault : ALIAS FOR ActuatorFault.Ack;   // 1=Actuator Fault Alarm has been acknowledged
   Sts_ActuatorFaultDisabled : ALIAS FOR ActuatorFault.Disabled;   // 1=Actuator Fault Alarm has been Disabled by Maintenance
   Sts_ActuatorFaultShelved : ALIAS FOR ActuatorFault.Shelved;   // 1=Actuator Fault Alarm has been Shelved by Operator
   Sts_ActuatorFaultSuppressed : ALIAS FOR ActuatorFault.Suppressed;   // 1=Actuator Fault Alarm has been Suppressed by Program
   Sts_IOFault : ALIAS FOR IOFault.Inp;   // 1=I/O Fault Status (0=OK, 1=Bad)
   Alm_IOFault : ALIAS FOR IOFault.Alm;   // 1=I/O Fault Alarm
   Ack_IOFault : ALIAS FOR IOFault.Ack;   // 1=I/O Fault Alarm has been acknowledged
   Sts_IOFaultDisabled : ALIAS FOR IOFault.Disabled;   // 1=I/O Fault Alarm has been Disabled by Maintenance
   Sts_IOFaultShelved : ALIAS FOR IOFault.Shelved;   // 1=I/O Fault Alarm has been Shelved by Operator
   Sts_IOFaultSuppressed : ALIAS FOR IOFault.Suppressed;   // 1=I/O Fault Alarm has been Suppressed by Program
   Rdy_BumpOpen : BOOL;   // 1=Ready to receive OCmd_BumpOpen (enables HMI button)
   Rdy_BumpClose : BOOL;   // 1=Ready to receive OCmd_BumpClose (enables HMI button)
   Rdy_Bypass : BOOL; {access Read Only}   // 1=Ready to receive OCmd_Bypass (enables HMI button)
   Rdy_Check : BOOL; {access Read Only}   // 1=Ready to receive OCmd_Check (enables HMI button)
   Rdy_Disable : BOOL; {access Read Only}   // 1=Ready to receive MCmd_Disable (enables HMI button)
   Rdy_Enable : BOOL; {access Read Only}   // 1=Ready to receive MCmd_Enable (enables HMI button)
   Rdy_Reset : BOOL; {access Read Only}   // 1=Ready to receive OCmd_Reset (enables HMI button)
   Rdy_ResetAckAll : BOOL; {access Read Only}   // 1=At least one Alarm or latched Shed condition requires Reset or Ack
   Rdy_CV : BOOL; {access Read Only}   // 1=Ready to receive OSet_CV (enables data entry field)
   Rdy_CVRoCLimInc : BOOL; {access Read Only}   // 1=Ready to receive OSet_CVRoCLimInc (enables data entry field)
   Rdy_CVRoCLimDec : BOOL; {access Read Only}   // 1=Ready to receive OSet_CVRoCLimDec (enables data entry field)
   P_ValveC : BOOL;   // Unique Parameter Name for auto - discovery
END_VAR
VAR
   Mode : P_Mode := (Cfg_PCmdClear := 1, Cfg_OvrdOverLock := 1, Rdy_OAcq := 1);   // Pulse Output Valve Mode Selection
   IOFault : P_Alarm := (Cfg_AckReqd := 1, Cfg_AllowShelve := 1, Cfg_AllowDisable := 1, Cfg_PCmdClear := 1, Cfg_Severity := 1000, Cfg_AlmMinOnT := 5, PCfg_AllowExist := 1, Ack := 1);   // I/O Fault Alarm
   IntlkTrip : P_Alarm := (Cfg_AckReqd := 1, Cfg_AllowShelve := 1, Cfg_AllowDisable := 1, Cfg_PCmdClear := 1, Cfg_Severity := 500, Cfg_AlmMinOnT := 5, PCfg_AllowExist := 1, Ack := 1);   // Interlock Trip Alarm
   Cfg_Tag : STRING_20 := 'P_ValveC';   // Tagname for display on HMI
   Cfg_Label : STRING_20 := 'Control Valve';   // Label for graphic symbol displayed on HMI
   Cfg_Desc : STRING_40 := 'Control Valve';   // Description for display on HMI
   Wrk_Notify : DINT; {access None}   // Buffer for building Val_Notify
   Wrk_Bypass : BOOL; {access None}   // Internal Bypassable Interlocks are Bypassed flag
   Wrk_Disabled : BOOL; {access None}   // Internal Pulse Output Valve Disabled status
   Cfg_EU : STRING_8 := '% Open';   // Engineering Units for display on HMI
   Wrk_CV : REAL; {access None}   // Working copy of Speed Reference (for limiting)
   Wrk_CVRoCLimInc : REAL; {access None}   // Selected CV Rate of Change Limit Increasing
   Wrk_CVSet : REAL; {access None}   // Final selected CV to feed to RoC Limiter
   Wrk_CVOut : REAL; {access None}   // Working value of CV after Rate Limiting
   Wrk_IntlkTripONS : BOOL; {access None}   // Interlock Tripped This Scan
   Wrk_ScanTime : REAL; {access None}   // Seconds since previous scan
   Wrk_StepInc : REAL; {access None}   // Amount to increase CV (to valve pulse logic) this scan for rate limiting
   Wrk_ScanT : TIMER := (PRE := 2147483647); {access None}   // Scan Timer (milliseconds, always runs)
   Inf_Tab : SINT;   // Tab to display (FTView ME)
   Wrk_Sts : SINT; {access None}   // Buffer for building Val_Sts
   Wrk_Fault : SINT; {access None}   // Buffer for building Val_Fault
   Wrk_SrcQ : SINT; {access None}   // Register for building Source / Quality enumeration
   ActuatorFault : P_Alarm := (Cfg_AckReqd := 1, Cfg_AllowShelve := 1, Cfg_AllowDisable := 1, Cfg_PCmdClear := 1, Cfg_Severity := 1000, Cfg_AlmMinOnT := 5, PCfg_AllowExist := 1, Ack := 1);   // Actuator Fault Alarm (based on Actuator Fault Input)
   Wrk_RealChkDINT : DINT; {access None}   // REAL tag bit pattern as a DINT to check for Inf / NaN
   Wrk_Close : BOOL; {access None}   // Internal Close output -- before Sim
   Wrk_Open : BOOL; {access None}   // Internal Open output -- before Sim
   Wrk_CycleT : TIMER := (PRE := 2147483647); {access None}   // Overall Cycle Timer for pulsed outputs
   Wrk_OKtoOpen : BOOL; {access None}   // OK to pulse Out_Open
   Wrk_OKtoClose : BOOL; {access None}   // OK to pulse Out_Close
   Wrk_OpenTime : REAL; {access None}   // Time to pulse Out_Open
   Wrk_CycleT_ms : DINT; {access None}   // Cycle Time in milliseconds (preset)
   Wrk_OpenTimePrev : DINT; {access None}   // Wrk_OpenTime from previous cycle
   Wrk_CloseTime : REAL; {access None}   // Time to pulse Out_Close
   Wrk_CloseTimePrev : REAL; {access None}   // Wrk_CloseTime from previous cycle
   Inf_Type : STRING_16 := 'P_ValveC'; {access Read Only}   // Must contain AOI name, used for HMI and Information S/W
   Wrk_OpenFdbk : BOOL; {access None}   // 1=LS Feedback shows valve confirmed open
   Wrk_ClosedFdbk : BOOL; {access None}   // 1=LS Feedback shows valve confirmed closed
   Wrk_StepDec : REAL; {access None}   // Amount to decrease CV (to valve pulse logic) this scan for rate limiting
   Wrk_CVRoCLimDec : REAL; {access None}   // Selected CV Rate of Change Limit Decreasing
   Wrk_BumpClose : BOOL; {access None}   // Operator Bump Close requested
   Wrk_BumpOpen : BOOL; {access None}   // Operator Bump Open requested
   Wrk_BumpingOpen : BOOL; {access None}   // Operator Bump Open actively pulsing Out_Open
   Wrk_BumpingClose : BOOL; {access None}   // Operator Bump Close actively pulsing Out_Close
   Wrk_CycleActive : BOOL; {access None}   // Outputs are cycling; wait for cycle to complete
   Inf_Lib : STRING_12 := 'RA-BAS'; {access Read Only}   // Display Library for Faceplate call-up
   Cfg_CVNavTag : STRING_NavTag;   // Tagname for destination of CV Navigation button
   Wrk_ShedIntlkCV : BOOL; {access None}   // Output CV being held at Interlock value
   Wrk_ShedHold : BOOL; {access None}   // Output CV being held at last good value
END_VAR

ROUTINE EnableInFalse   (* ladder *)
// Disabled is asserted, Output OFF (zero), Alarms disabled
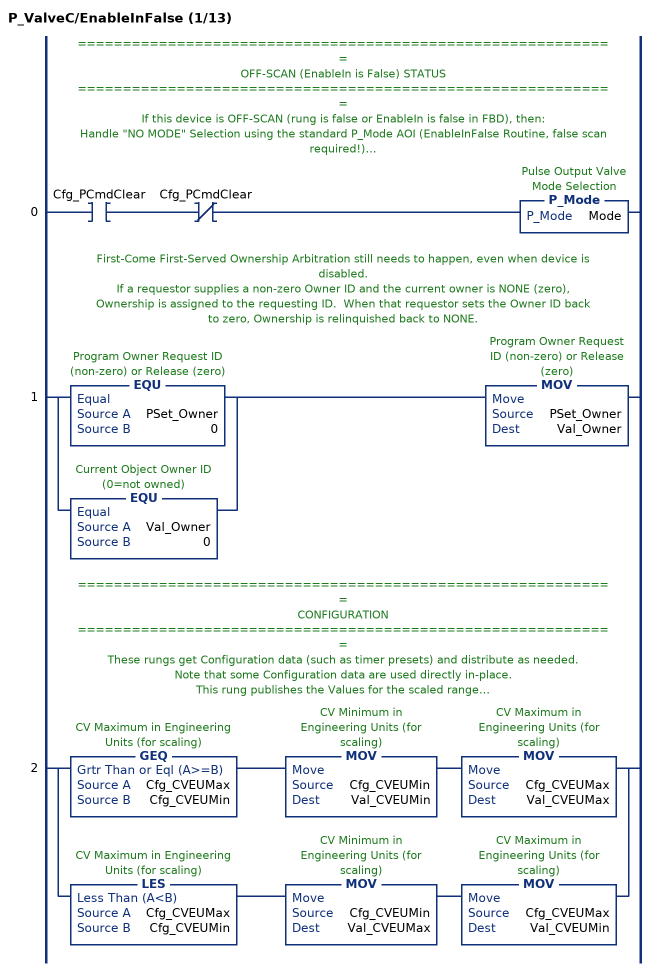
   // ============================================================
   // OFF-SCAN (EnableIn is False) STATUS
   // ============================================================
   // If this device is OFF-SCAN (rung is false or EnableIn is false in FBD), then:
   // Handle "NO MODE" Selection using the standard P_Mode AOI (EnableInFalse Routine, false scan required!).
   // NOTE:  IN ORDER TO AVOID USING AN "AFI" (which will generate a routine verify warning),
   // THIS RUNG USES AN XIC of Cfg_PCmdClear, followed by an XIO of the SAME BIT
   // to ensure P_Mode is SCANNED FALSE ("NO MODE").
   // THIS IS NOT DEAD CODE AND MUST APPEAR EXACTLY AS SHOWN FOR PROPER OPERATION!
   0: XIC(Cfg_PCmdClear)XIO(Cfg_PCmdClear)P_Mode(Mode);
   // First-Come First-Served Ownership Arbitration still needs to happen, even when device is disabled.
   // If a requestor supplies a non-zero Owner ID and the current owner is NONE (zero),
   // Ownership is assigned to the requesting ID.  When that requestor sets the Owner ID back
   // to zero, Ownership is relinquished back to NONE.
   1: [EQU(PSet_Owner,0) ,EQU(Val_Owner,0) ]MOV(PSet_Owner,Val_Owner);
   // ============================================================
   // CONFIGURATION
   // ============================================================
   // These rungs get Configuration data (such as timer presets) and distribute as needed.
   // Note that some Configuration data are used directly in-place.
   // This rung publishes the Values for the scaled range.
   // If this instruction is reverse scaled by reversing the scaled (EU) min and max configurations,
   // the values are swapped so the the EUMax Value is always greater than the EUMin Value.
   // This makes the HMI bargraph and trend coding easier, and provides values
   // that can be pinned to the CV EU configuration of a PID, so the AOut and PID ranges are in lockstep.
   2: [GEQ(Cfg_CVEUMax,Cfg_CVEUMin) MOV(Cfg_CVEUMin,Val_CVEUMin) MOV(Cfg_CVEUMax,Val_CVEUMax) ,LES(Cfg_CVEUMax,Cfg_CVEUMin) MOV(Cfg_CVEUMin,Val_CVEUMax) MOV(Cfg_CVEUMax,Val_CVEUMin) ];
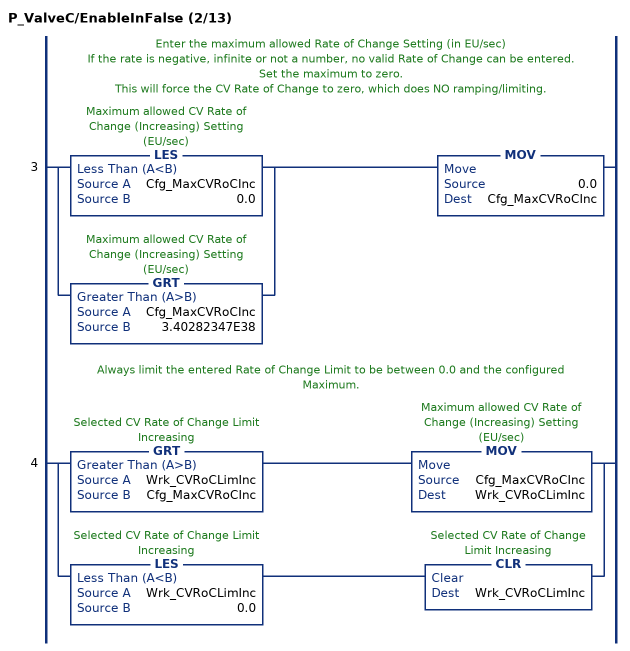
   // Enter the maximum allowed Rate of Change Setting (in EU/sec)
   // If the rate is negative, infinite or not a number, no valid Rate of Change can be entered.  Set the maximum to zero.
   // This will force the CV Rate of Change to zero, which does NO ramping/limiting.
   3: [LES(Cfg_MaxCVRoCInc,0.0) ,GRT(Cfg_MaxCVRoCInc,3.40282347E38) ]MOV(0.0,Cfg_MaxCVRoCInc);
   // Always limit the entered Rate of Change Limit to be between 0.0 and the configured Maximum.
   4: [GRT(Wrk_CVRoCLimInc,Cfg_MaxCVRoCInc) MOV(Cfg_MaxCVRoCInc,Wrk_CVRoCLimInc) ,LES(Wrk_CVRoCLimInc,0.0) CLR(Wrk_CVRoCLimInc) ];
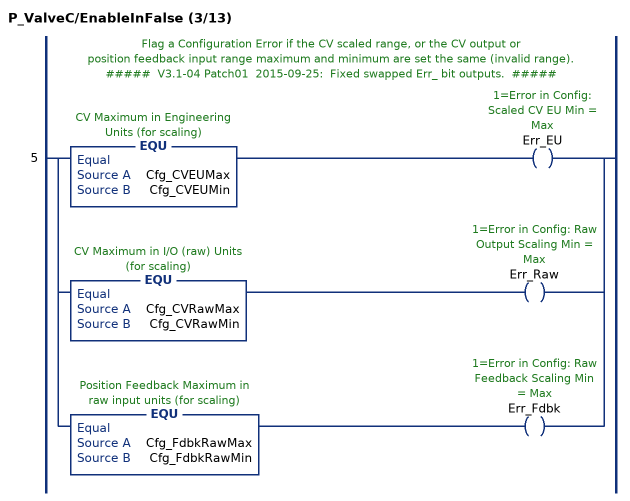
   // Flag a Configuration Error if the CV scaled range, or the CV output or
   // position feedback input range maximum and minimum are set the same (invalid range).
   // #####  V3.1-04 Patch01  2015-09-25:  Fixed swapped Err_ bit outputs.  #####
   5: [EQU(Cfg_CVEUMax,Cfg_CVEUMin) OTE(Err_EU) ,EQU(Cfg_CVRawMax,Cfg_CVRawMin) OTE(Err_Raw) ,EQU(Cfg_FdbkRawMax,Cfg_FdbkRawMin) OTE(Err_Fdbk) ];
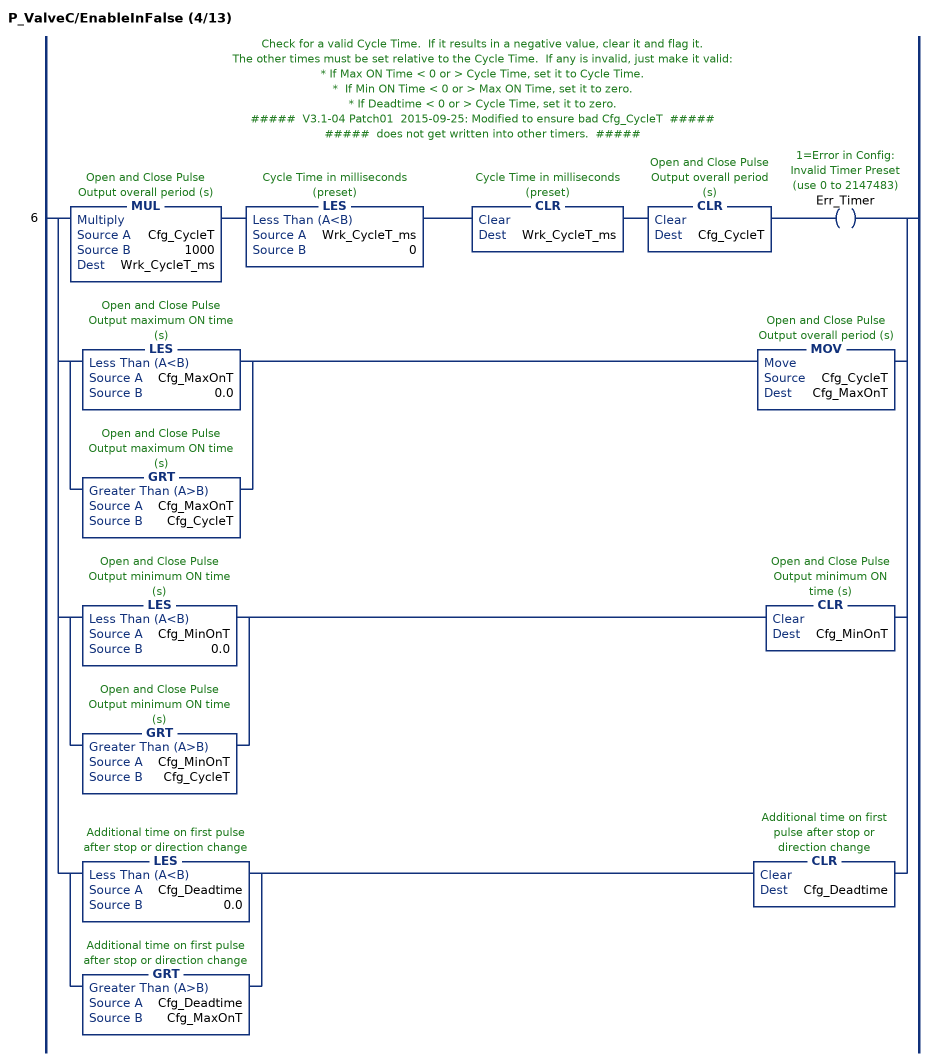
   // Check for a valid Cycle Time.  If it results in a negative value, clear it and flag it.
   // The other times must be set relative to the Cycle Time.  If any is invalid, just make it valid:
   // * If Max ON Time < 0 or > Cycle Time, set it to Cycle Time.
   // *  If Min ON Time < 0 or > Max ON Time, set it to zero.
   // * If Deadtime < 0 or > Cycle Time, set it to zero.
   // #####  V3.1-04 Patch01  2015-09-25: Modified to ensure bad Cfg_CycleT  #####
   // #####  does not get written into other timers.  #####
   6: [MUL(Cfg_CycleT,1000,Wrk_CycleT_ms) LES(Wrk_CycleT_ms,0) CLR(Wrk_CycleT_ms) CLR(Cfg_CycleT) OTE(Err_Timer) ,[LES(Cfg_MaxOnT,0.0) ,GRT(Cfg_MaxOnT,Cfg_CycleT) ] MOV(Cfg_CycleT,Cfg_MaxOnT) ,[LES(Cfg_MinOnT,0.0) ,GRT(Cfg_MinOnT,Cfg_CycleT) ] CLR(Cfg_MinOnT) ,[LES(Cfg_Deadtime,0.0) ,GRT(Cfg_Deadtime,Cfg_MaxOnT) ] CLR(Cfg_Deadtime) ];
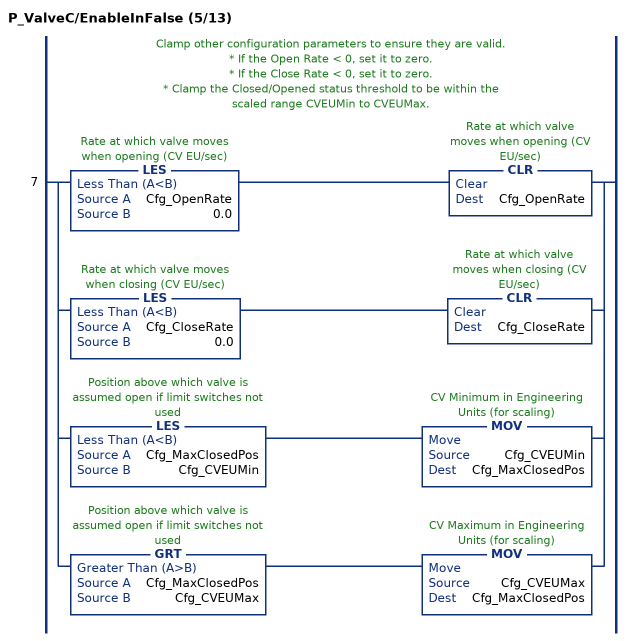
   // Clamp other configuration parameters to ensure they are valid.
   // * If the Open Rate < 0, set it to zero.
   // * If the Close Rate < 0, set it to zero.
   // * Clamp the Closed/Opened status threshold to be within the
   // scaled range CVEUMin to CVEUMax.
   7: [LES(Cfg_OpenRate,0.0) CLR(Cfg_OpenRate) ,LES(Cfg_CloseRate,0.0) CLR(Cfg_CloseRate) ,LES(Cfg_MaxClosedPos,Cfg_CVEUMin) MOV(Cfg_CVEUMin,Cfg_MaxClosedPos) ,GRT(Cfg_MaxClosedPos,Cfg_CVEUMax) MOV(Cfg_CVEUMax,Cfg_MaxClosedPos) ];
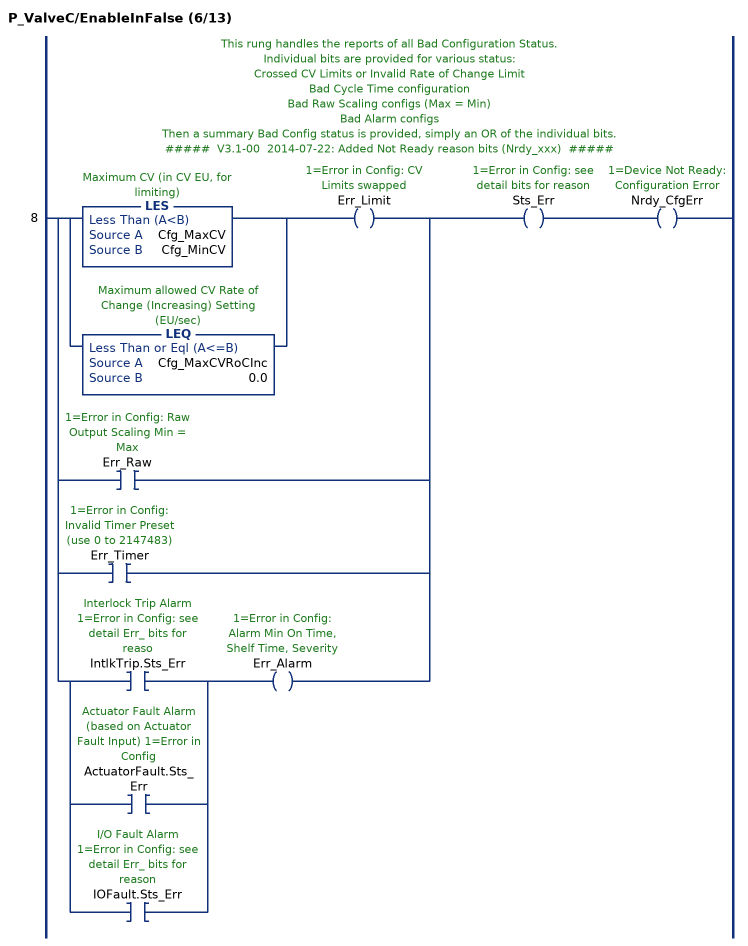
   // This rung handles the reports of all Bad Configuration Status.
   // Individual bits are provided for various status:
   // Crossed CV Limits or Invalid Rate of Change Limit
   // Bad Cycle Time configuration
   // Bad Raw Scaling configs (Max = Min)
   // Bad Alarm configs
   // Then a summary Bad Config status is provided, simply an OR of the individual bits.
   // #####  V3.1-00  2014-07-22: Added Not Ready reason bits (Nrdy_xxx)  #####
   8: [[LES(Cfg_MaxCV,Cfg_MinCV) ,LEQ(Cfg_MaxCVRoCInc,0.0) ] OTE(Err_Limit) ,XIC(Err_Raw) ,XIC(Err_Timer) ,[XIC(IntlkTrip.Sts_Err) ,XIC(ActuatorFault.Sts_Err) ,XIC(IOFault.Sts_Err) ] OTE(Err_Alarm) ]OTE(Sts_Err)OTE(Nrdy_CfgErr);
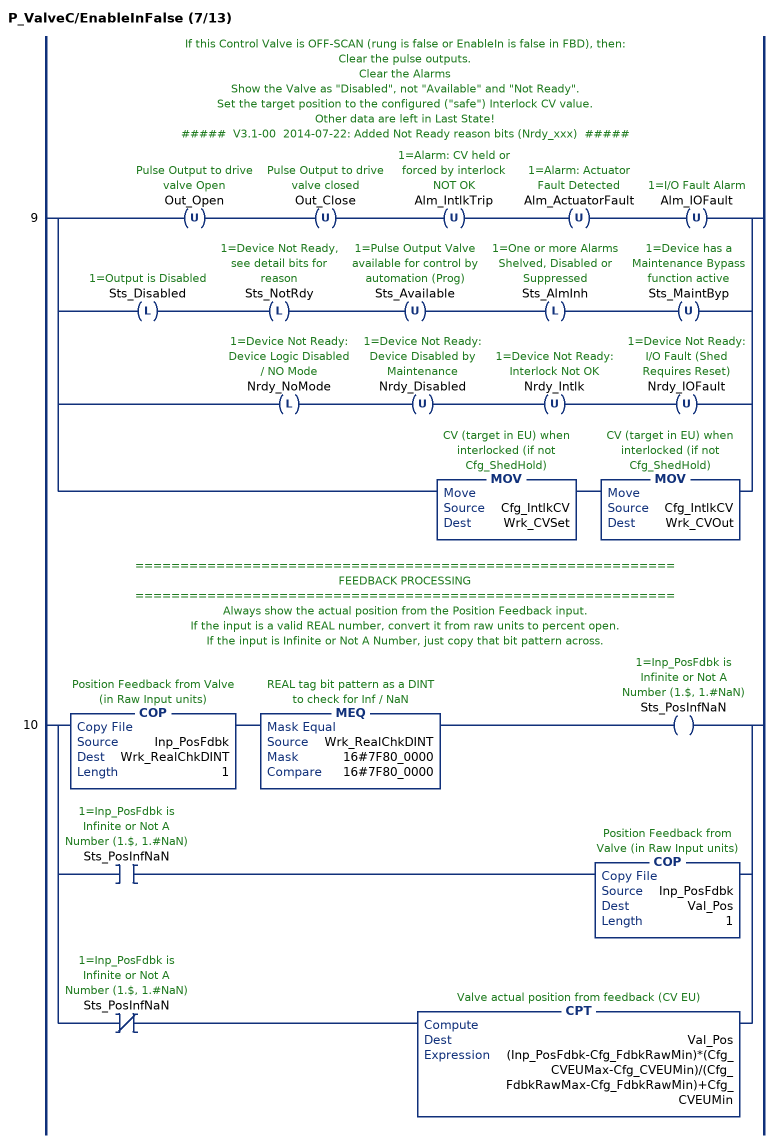
   // If this Control Valve is OFF-SCAN (rung is false or EnableIn is false in FBD), then:
   // Clear the pulse outputs.
   // Clear the Alarms
   // Show the Valve as "Disabled", not "Available" and "Not Ready".
   // Set the target position to the configured ("safe") Interlock CV value.
   // Other data are left in Last State!
   // #####  V3.1-00  2014-07-22: Added Not Ready reason bits (Nrdy_xxx)  #####
   9: [OTU(Out_Open) OTU(Out_Close) OTU(Alm_IntlkTrip) OTU(Alm_ActuatorFault) OTU(Alm_IOFault) ,OTL(Sts_Disabled) OTL(Sts_NotRdy) OTU(Sts_Available) OTL(Sts_AlmInh) OTU(Sts_MaintByp) ,OTL(Nrdy_NoMode) OTU(Nrdy_Disabled) OTU(Nrdy_Intlk) OTU(Nrdy_IOFault) ,MOV(Cfg_IntlkCV,Wrk_CVSet) MOV(Cfg_IntlkCV,Wrk_CVOut) ];
   // ============================================================
   // FEEDBACK PROCESSING
   // ============================================================
   // Always show the actual position from the Position Feedback input.
   // If the input is a valid REAL number, convert it from raw units to percent open.
   // If the input is Infinite or Not A Number, just copy that bit pattern across.
   10: [COP(Inp_PosFdbk,Wrk_RealChkDINT,1) MEQ(Wrk_RealChkDINT,16#7F80_0000,16#7F80_0000) OTE(Sts_PosInfNaN) ,XIC(Sts_PosInfNaN) COP(Inp_PosFdbk,Val_Pos,1) ,XIO(Sts_PosInfNaN) CPT(Val_Pos,(Inp_PosFdbk-Cfg_FdbkRawMin)*(Cfg_CVEUMax-Cfg_CVEUMin)/(Cfg_FdbkRawMax-Cfg_FdbkRawMin)+Cfg_CVEUMin) ];
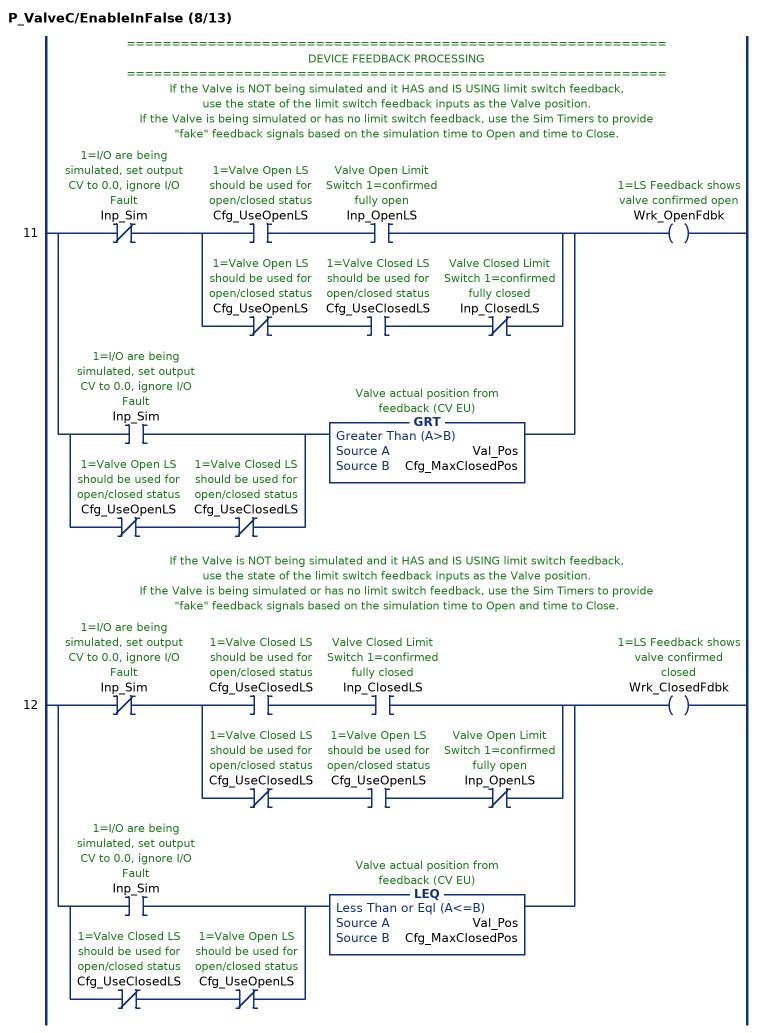
   // ============================================================
   // DEVICE FEEDBACK PROCESSING
   // ============================================================
   // If the Valve is NOT being simulated and it HAS and IS USING limit switch feedback,
   // use the state of the limit switch feedback inputs as the Valve position.
   // If the Valve is being simulated or has no limit switch feedback, use the Sim Timers to provide
   // "fake" feedback signals based on the simulation time to Open and time to Close.
   11: [XIO(Inp_Sim) [XIC(Cfg_UseOpenLS) XIC(Inp_OpenLS) ,XIO(Cfg_UseOpenLS) XIC(Cfg_UseClosedLS) XIO(Inp_ClosedLS) ] ,[XIC(Inp_Sim) ,XIO(Cfg_UseOpenLS) XIO(Cfg_UseClosedLS) ] GRT(Val_Pos,Cfg_MaxClosedPos) ]OTE(Wrk_OpenFdbk);
   // If the Valve is NOT being simulated and it HAS and IS USING limit switch feedback,
   // use the state of the limit switch feedback inputs as the Valve position.
   // If the Valve is being simulated or has no limit switch feedback, use the Sim Timers to provide
   // "fake" feedback signals based on the simulation time to Open and time to Close.
   12: [XIO(Inp_Sim) [XIC(Cfg_UseClosedLS) XIC(Inp_ClosedLS) ,XIO(Cfg_UseClosedLS) XIC(Cfg_UseOpenLS) XIO(Inp_OpenLS) ] ,[XIC(Inp_Sim) ,XIO(Cfg_UseClosedLS) XIO(Cfg_UseOpenLS) ] LEQ(Val_Pos,Cfg_MaxClosedPos) ]OTE(Wrk_ClosedFdbk);
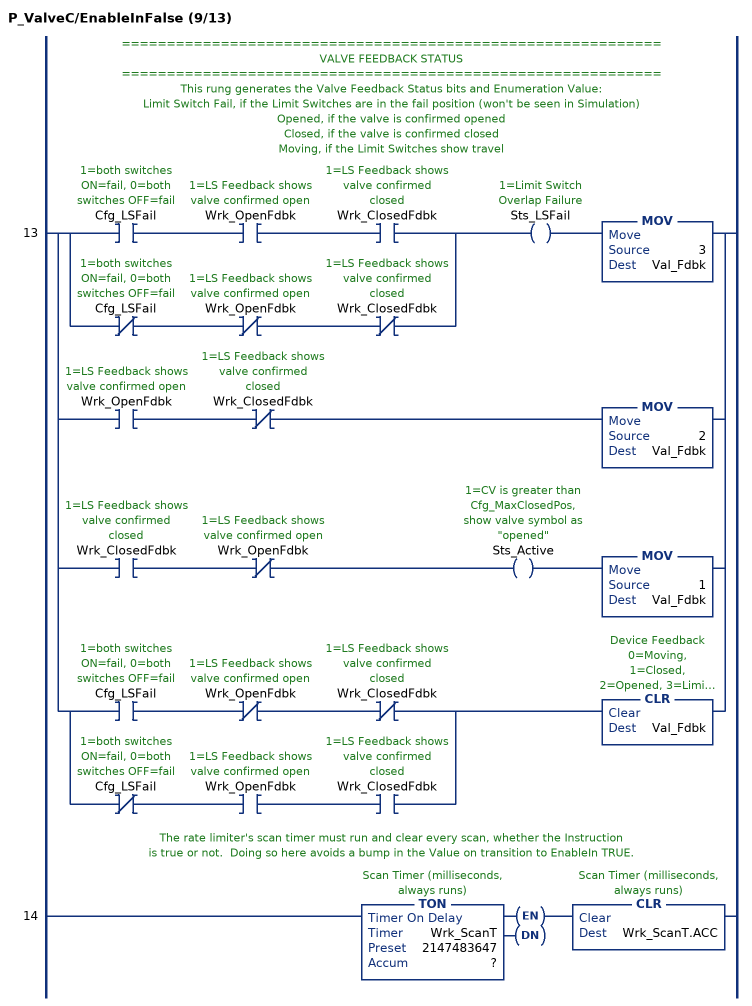
   // ============================================================
   // VALVE FEEDBACK STATUS
   // ============================================================
   // This rung generates the Valve Feedback Status bits and Enumeration Value:
   // Limit Switch Fail, if the Limit Switches are in the fail position (won't be seen in Simulation)
   // Opened, if the valve is confirmed opened
   // Closed, if the valve is confirmed closed
   // Moving, if the Limit Switches show travel
   13: [[XIC(Cfg_LSFail) XIC(Wrk_OpenFdbk) XIC(Wrk_ClosedFdbk) ,XIO(Cfg_LSFail) XIO(Wrk_OpenFdbk) XIO(Wrk_ClosedFdbk) ] OTE(Sts_LSFail) MOV(3,Val_Fdbk) ,XIC(Wrk_OpenFdbk) XIO(Wrk_ClosedFdbk) MOV(2,Val_Fdbk) ,XIC(Wrk_ClosedFdbk) XIO(Wrk_OpenFdbk) OTE(Sts_Active) MOV(1,Val_Fdbk) ,[XIC(Cfg_LSFail) XIO(Wrk_OpenFdbk) XIO(Wrk_ClosedFdbk) ,XIO(Cfg_LSFail) XIC(Wrk_OpenFdbk) XIC(Wrk_ClosedFdbk) ] CLR(Val_Fdbk) ];
   // The rate limiter's scan timer must run and clear every scan, whether the Instruction
   // is true or not.  Doing so here avoids a bump in the Value on transition to EnableIn TRUE.
   14: TON(Wrk_ScanT,?,?)CLR(Wrk_ScanT.ACC);
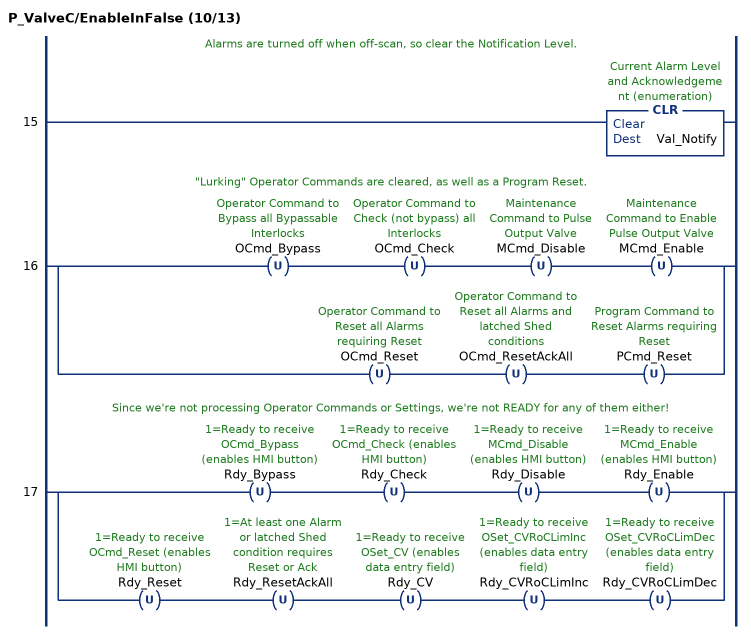
   // Alarms are turned off when off-scan, so clear the Notification Level.
   15: CLR(Val_Notify);
   // "Lurking" Operator Commands are cleared, as well as a Program Reset.
   16: [OTU(OCmd_Bypass) OTU(OCmd_Check) OTU(MCmd_Disable) OTU(MCmd_Enable) ,OTU(OCmd_Reset) OTU(OCmd_ResetAckAll) OTU(PCmd_Reset) ];
   // Since we're not processing Operator Commands or Settings, we're not READY for any of them either!
   17: [OTU(Rdy_Bypass) OTU(Rdy_Check) OTU(Rdy_Disable) OTU(Rdy_Enable) ,OTU(Rdy_Reset) OTU(Rdy_ResetAckAll) OTU(Rdy_CV) OTU(Rdy_CVRoCLimInc) OTU(Rdy_CVRoCLimDec) ];
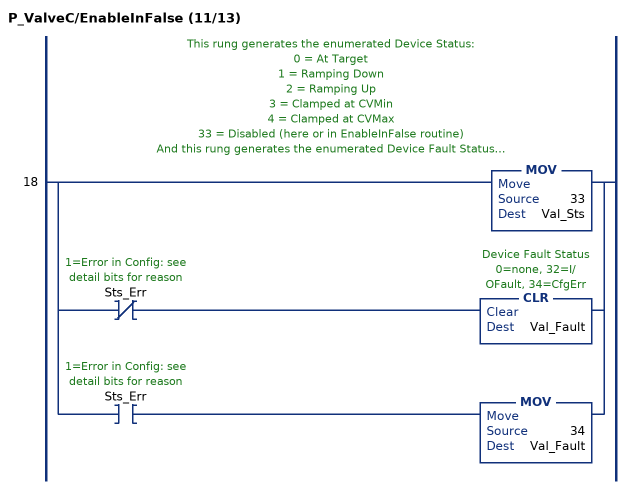
   // This rung generates the enumerated Device Status:
   // 0 = At Target
   // 1 = Ramping Down
   // 2 = Ramping Up
   // 3 = Clamped at CVMin
   // 4 = Clamped at CVMax
   // 33 = Disabled (here or in EnableInFalse routine)
   // And this rung generates the enumerated Device Fault Status:
   // 0 = none
   // 32 = I/O Fault
   // 34 = Configuration Error
   18: [MOV(33,Val_Sts) ,XIO(Sts_Err) CLR(Val_Fault) ,XIC(Sts_Err) MOV(34,Val_Fault) ];
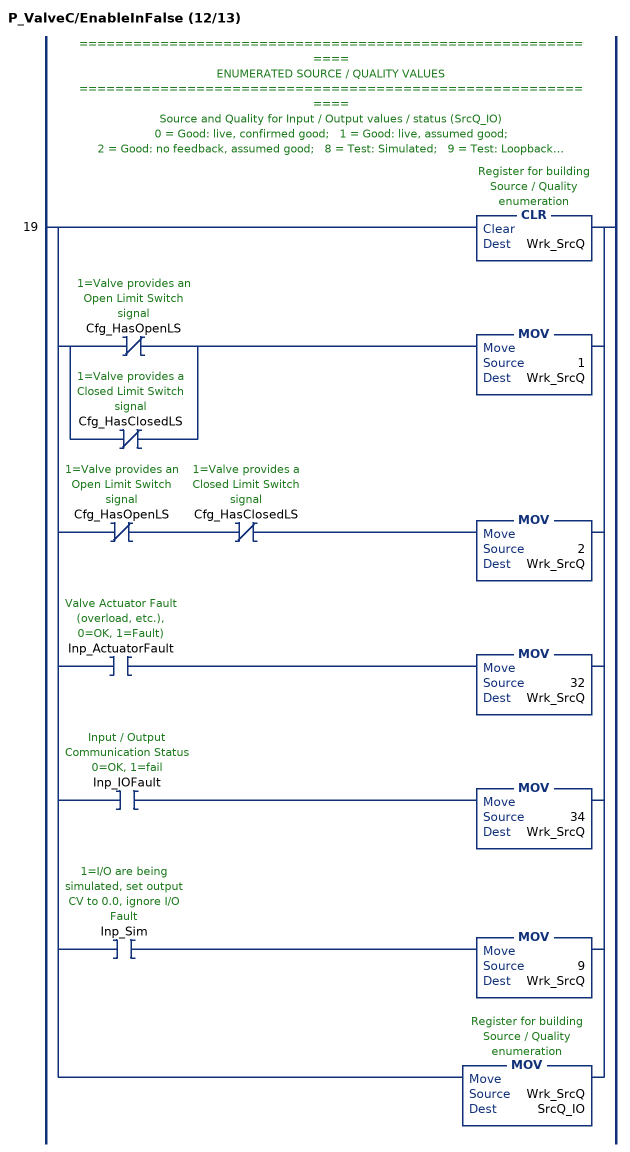
   // ============================================================
   // ENUMERATED SOURCE / QUALITY VALUES
   // ============================================================
   // Source and Quality for Input / Output values / status (SrcQ_IO)
   // 0 = Good: live, confirmed good;   1 = Good: live, assumed good;
   // 2 = Good: no feedback, assumed good;   8 = Test: Simulated;   9 = Test: Loopback;
   // 10 = Test: Manually Entered;   16 = Uncertain: Live, off-spec;
   // 17 = Uncertain, Substituted at Device / Bus;   18 = Uncertain, Substituted at AOI;
   // 19 = Uncertain, using last known good;    20 = Uncertain, using replacement value;
   // 32 = Bad, Signal Failure;   33 = Bad, Channel Fault;
   // 34 = Bad, Module / Comms Fault;   35 = Bad, Invalid Configuration
   // #####  V3.1-00  2014-07-22:  Added rung for Source/Quality enumerations.  #####
   19: [CLR(Wrk_SrcQ) ,[XIO(Cfg_HasOpenLS) ,XIO(Cfg_HasClosedLS) ] MOV(1,Wrk_SrcQ) ,XIO(Cfg_HasOpenLS) XIO(Cfg_HasClosedLS) MOV(2,Wrk_SrcQ) ,XIC(Inp_ActuatorFault) MOV(32,Wrk_SrcQ) ,XIC(Inp_IOFault) MOV(34,Wrk_SrcQ) ,XIC(Inp_Sim) MOV(9,Wrk_SrcQ) ,MOV(Wrk_SrcQ,SrcQ_IO) ];
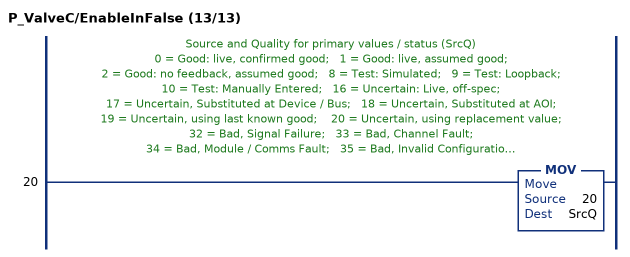
   // Source and Quality for primary values / status (SrcQ)
   // 0 = Good: live, confirmed good;   1 = Good: live, assumed good;
   // 2 = Good: no feedback, assumed good;   8 = Test: Simulated;   9 = Test: Loopback;
   // 10 = Test: Manually Entered;   16 = Uncertain: Live, off-spec;
   // 17 = Uncertain, Substituted at Device / Bus;   18 = Uncertain, Substituted at AOI;
   // 19 = Uncertain, using last known good;    20 = Uncertain, using replacement value;
   // 32 = Bad, Signal Failure;   33 = Bad, Channel Fault;
   // 34 = Bad, Module / Comms Fault;   35 = Bad, Invalid Configuration
   // #####  V3.1-00  2014-07-22:  Added rung for Source/Quality enumerations.  #####
   20: MOV(20,SrcQ);
END_ROUTINE
